FUNCTION_BLOCK FB_Bel_Lichtsensor
VAR_INPUT
END_VAR
VAR_OUTPUT
	Helligkeit				: REAL;
END_VAR
VAR
	IN_Helligkeit 		AT %I* 	: INT;
	VAR_Helligkeit				: REAL;
END_VAR

VAR_Helligkeit := IN_Helligkeit;
Helligkeit	:= (32767 - VAR_Helligkeit)/13.71 + 10 ; (* gibt die Helligkeit in Lux, laut Sensor-Datasheet*)

END_FUNCTION_BLOCK

(* stored: Version 1.1.0.1, ProductVersion 3.1.4024.9
   POU FB_Bel_Lichtsensor: Id {a3310165-f3c5-4134-bb94-4ae1086b22f9}, SpecialFunc None *)
